{attribute 'qualified_only' := ''}
{attribute 'strict' := ''}
TYPE AXIS_DIRECTION :
(
	DirectionPositive := 0,
	DirectionNegative := 1
);
END_TYPE

(* stored: Version 1.1.0.1, ProductVersion 3.1.4024.12
   DUT AXIS_DIRECTION: Id {1651d020-cb9b-412f-bbbc-1fc04036f18d} *)
